// TIA Portal project "StartStopMotore" (V20)
// Si andrà a realizzare un programma che
// consentirà di simulare un’operazione di marcia e
// arresto di un motore industriale.

(* hardware
DEVICE "S7-1200 station_1"  S7-1200 Station
   slot 0: "Rack_0"  S7-1200 Rack  Rack  V1.0
   slot 1: "Playground_PLC"  CPU 1214C DC/DC/DC  6ES7 214-1AG40-0XB0  V4.7
   slot 3: "AQ 1x12BIT_1"  AQ1 signal board  6ES7 232-4HA30-0XB0  V1.0
*)

// ===== PLC "Playground_PLC"  CPU 1214C DC/DC/DC =====

DATA_BLOCK "MOTORE"   // DB2
{ S7_Optimized_Access := 'TRUE' }
VERSION : 0.1
   VAR
      START : Bool;
      STOP : Bool;
      MOTORE : Bool;
   END_VAR
BEGIN
END_DATA_BLOCK

ORGANIZATION_BLOCK "Main"   // OB1, LAD, ProgramCycle
TITLE = "Main Program Sweep (Cycle)"
{ S7_Optimized_Access := 'TRUE' }
VERSION : 0.1
   VAR_INPUT
      Initial_Call : Bool;   // Initial call of this OB
      Remanence : Bool;   // =True, if remanent data are available
   END_VAR
BEGIN

REGION Network 1
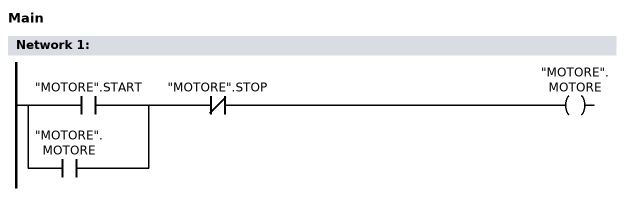
   RUNG wire#powerrail
      Contact( "MOTORE".START )
      wire#w1
      I_Contact( "MOTORE".STOP )
      Coil( "MOTORE".MOTORE )
   END_RUNG
   RUNG wire#powerrail
      Contact( "MOTORE".MOTORE )
   END_RUNG wire#w1
   // the same network as SCL:
   "MOTORE".MOTORE := ("MOTORE".START OR "MOTORE".MOTORE) AND NOT "MOTORE".STOP;
END_REGION
END_ORGANIZATION_BLOCK